FUNCTION_BLOCK FB_Messenger
VAR_INPUT
END_VAR
VAR_OUTPUT
END_VAR
VAR
END_VAR

{attribute 'TcRpcEnable'}
METHOD Send : LREAL
VAR_INPUT
	stMessage_Info 	: ST_MESSAGE_INFO;
	arfData 		: ARRAY[0..2] OF LREAL;
END_VAR
VAR_OUTPUT
	sReturn_Message : WSTRING;
	bSuccess 		: BOOL; 
END_VAR
VAR_INST 
	stMessage_Info_Copy : ST_MESSAGE_INFO;
	arfData_Copy : ARRAY[0..2] OF LREAL;
END_VAR
VAR 
	i : DINT;
END_VAR
stMessage_Info_Copy := stMessage_Info;
arfData_Copy 		:= arfData;

CASE stMessage_Info.eOperation OF
	E_OPERATION.Array_Sum:
		FOR i := 0 TO SIZEOF(arfDATA)/SIZEOF(arfData[0])-1 DO
			Send := Send + arfData[i];
			END_FOR
	E_OPERATION.Array_Product:
		Send := arfData[0];
		FOR i := 1 TO SIZEOF(arfDATA)/SIZEOF(arfData[0])-1 DO
			Send := Send * arfData[i];
			END_FOR
END_CASE

sReturn_Message := "I have finished!";
bSuccess 		:= TRUE;
END_METHOD

END_FUNCTION_BLOCK

(* stored: Version 1.1.0.1, ProductVersion 3.1.4024.12
   POU FB_Messenger: Id {0b3bada7-ec5d-4f4b-8471-76143af8631b}, SpecialFunc None
   Method Send: Id {e0ce973a-a0de-43db-a81c-34c15d492236} *)
